// TIA Portal V17 export
// export: Created 2023-12-22T15:08:10.2331174Z, ExportSetting WithDefaults, DisplayName Totally Integrated Automation Portal, DisplayVersion V17, DisplayName TIA Portal Openness, DisplayVersion V17, DisplayName TIA Portal Version Control Interface, DisplayVersion V17, DisplayName STEP 7 Professional, DisplayVersion V17, DisplayName STEP 7 Safety, DisplayVersion V17, DisplayName WinCC Advanced, DisplayVersion V17
DATA_BLOCK "PS_StartUp_DB"   // DB13
VERSION : 0.1
// stored: AutoNumber false, DBAccessibleFromOPCUA true, DBAccessibleFromWebserver true, InstanceOfName PS_StartUp, InstanceOfType FB
"PS_StartUp"
   // VAR_INPUT
   //    PE : Real;
   //    LE_Target : Real;
   //    LE_Source : Real;
   // END_VAR
   // VAR_IN_OUT
   //    REQ : Int;
   //    Hz : Real;
   // END_VAR
   // VAR RETAIN
   //    Start : Bool;
   //    Ready : Bool;
   //    "Step" : Int;
   //    Warning : Word;
   //    PE_Point : Real;
   //    PE_Delta : Real;
   //    PE_Min : Real;
   //    LE_Target_Point : Real;
   //    LE_Target_Delta : Real;
   //    LE_Target_Min : Real;
   //    LE_Source_Point : Real;
   //    LE_Source_Delta : Real;
   //    LE_Source_Min : Real;
   //    xSP : Array[0..5] of Struct
   //       Use { S7_SetPoint := 'True'} : Bool;
   //       REQ { S7_SetPoint := 'True'} : Int;
   //       Hz { S7_SetPoint := 'True'} : Real;
   //       PE { S7_SetPoint := 'True'} : Real;
   //       PE_Delta : Real;
   //    END_STRUCT;
   //    xTime { S7_SetPoint := 'True'} : Array[0..5] of "Time_M";
   // END_VAR
BEGIN
   xSP[0..5].Use := TRUE;
   xSP[0].REQ := 1;
   xSP[1].REQ := 2;
   xSP[2].REQ := 3;
   xSP[3..5].REQ := 4;
   xSP[0].Hz := 36.0;
   xSP[1..2].Hz := 38.0;
   xSP[3].Hz := 40.0;
   xSP[4].Hz := 42.0;
   xSP[5].Hz := 44.0;
   xSP[0..1].PE := 5.0;
   xSP[2].PE := 6.0;
   xSP[3].PE := 6.5;
   xSP[4].PE := 7.0;
   xSP[5].PE := 10.0;
   xTime[0..1].SP_M := 5;
   xTime[2].SP_M := 1;
   xTime[3..5].SP_M := 0;
   xTime[0..1].SP_S := 0;
   xTime[2..5].SP_S := 30;
END_DATA_BLOCK
